(* IEC 61131-3 sources: mastertool-rankine-bridge/tests/indexer/fixtures/sample_export/objects/application_fb_2__FB_TimerSintetico, 1 file *)

(* ---- declaration.st ---- *)
FUNCTION_BLOCK FB_TimerSintetico
VAR_INPUT
    xStart          : BOOL;
END_VAR
VAR_IN_OUT
    tPreset         : TIME;
END_VAR
VAR_OUTPUT
    xDone           : BOOL;
END_VAR
